% RSLogix 500 project MLO3B JOB 15.RSS, saved by version 10.00.00.00 %
PROJECT "MLO3B"    % processor: Bul.1763 MicroLogix 1100 Series B %

PROGRAM FILES
  LAD 2   15 rungs

DATA FILES
  O0 OUTPUT  4 elements
  I1 INPUT  6 elements
  S2 STATUS  66 elements
  B3 BINARY  1 elements
  T4 TIMER  1 elements
  C5 COUNTER  1 elements
  R6 CONTROL  1 elements
  N7 INTEGER  1 elements
  F8 FLOAT  1 elements

LADDER 2
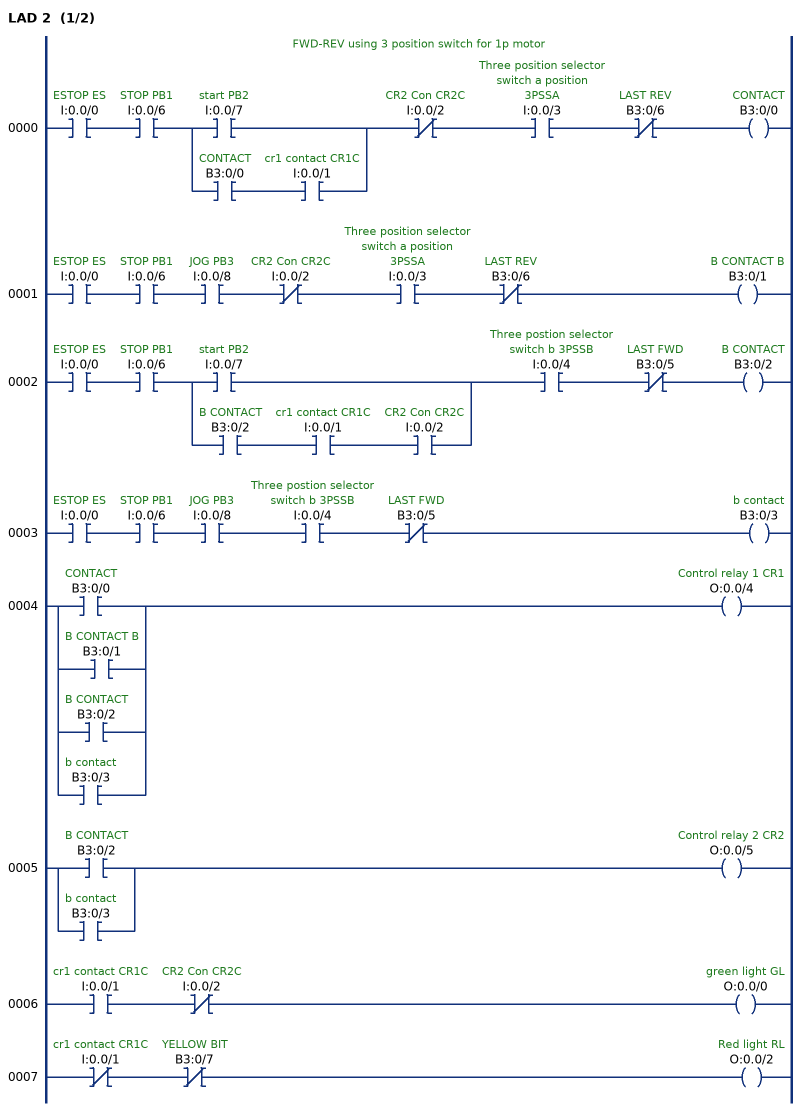
% Rung: 0 %
% FWD-REV using 3 position switch for 1p motor %
SOR XIC I:0.0/0 XIC I:0.0/6 BST XIC I:0.0/7 NXB XIC B3:0/0 XIC I:0.0/1 BND XIO I:0.0/2 XIC I:0.0/3 XIO B3:0/6 OTE B3:0/0 EOR
%   I:0.0/0  ES  "ESTOP" %
%   I:0.0/6  PB1  "STOP" %
%   I:0.0/7  PB2  "start" %
%   B3:0/0  CONTACT %
%   I:0.0/1  CR1C  "cr1 contact" %
%   I:0.0/2  CR2C  "CR2 Con" %
%   I:0.0/3  3PSSA  "Three position selector switch a position" %
%   B3:0/6  "LAST REV" %
% Rung: 1 %
SOR XIC I:0.0/0 XIC I:0.0/6 XIC I:0.0/8 XIO I:0.0/2 XIC I:0.0/3 XIO B3:0/6 OTE B3:0/1 EOR
%   I:0.0/0  ES  "ESTOP" %
%   I:0.0/6  PB1  "STOP" %
%   I:0.0/8  PB3  "JOG" %
%   I:0.0/2  CR2C  "CR2 Con" %
%   I:0.0/3  3PSSA  "Three position selector switch a position" %
%   B3:0/6  "LAST REV" %
%   B3:0/1  B  "B CONTACT" %
% Rung: 2 %
SOR XIC I:0.0/0 XIC I:0.0/6 BST XIC I:0.0/7 NXB XIC B3:0/2 XIC I:0.0/1 XIC I:0.0/2 BND XIC I:0.0/4 XIO B3:0/5 OTE B3:0/2 EOR
%   I:0.0/0  ES  "ESTOP" %
%   I:0.0/6  PB1  "STOP" %
%   I:0.0/7  PB2  "start" %
%   B3:0/2  "B CONTACT" %
%   I:0.0/1  CR1C  "cr1 contact" %
%   I:0.0/2  CR2C  "CR2 Con" %
%   I:0.0/4  3PSSB  "Three postion selector switch b" %
%   B3:0/5  "LAST FWD" %
% Rung: 3 %
SOR XIC I:0.0/0 XIC I:0.0/6 XIC I:0.0/8 XIC I:0.0/4 XIO B3:0/5 OTE B3:0/3 EOR
%   I:0.0/0  ES  "ESTOP" %
%   I:0.0/6  PB1  "STOP" %
%   I:0.0/8  PB3  "JOG" %
%   I:0.0/4  3PSSB  "Three postion selector switch b" %
%   B3:0/5  "LAST FWD" %
%   B3:0/3  "b contact" %
% Rung: 4 %
SOR BST XIC B3:0/0 NXB XIC B3:0/1 NXB XIC B3:0/2 NXB XIC B3:0/3 BND OTE O:0.0/4 EOR
%   B3:0/0  CONTACT %
%   B3:0/1  B  "B CONTACT" %
%   B3:0/2  "B CONTACT" %
%   B3:0/3  "b contact" %
%   O:0.0/4  CR1  "Control relay 1" %
% Rung: 5 %
SOR BST XIC B3:0/2 NXB XIC B3:0/3 BND OTE O:0.0/5 EOR
%   B3:0/2  "B CONTACT" %
%   B3:0/3  "b contact" %
%   O:0.0/5  CR2  "Control relay 2" %
% Rung: 6 %
SOR XIC I:0.0/1 XIO I:0.0/2 OTE O:0.0/0 EOR
%   I:0.0/1  CR1C  "cr1 contact" %
%   I:0.0/2  CR2C  "CR2 Con" %
%   O:0.0/0  GL  "green light" %
% Rung: 7 %
SOR XIO I:0.0/1 XIO B3:0/7 OTE O:0.0/2 EOR
%   I:0.0/1  CR1C  "cr1 contact" %
%   B3:0/7  "YELLOW BIT" %
%   O:0.0/2  RL  "Red light" %

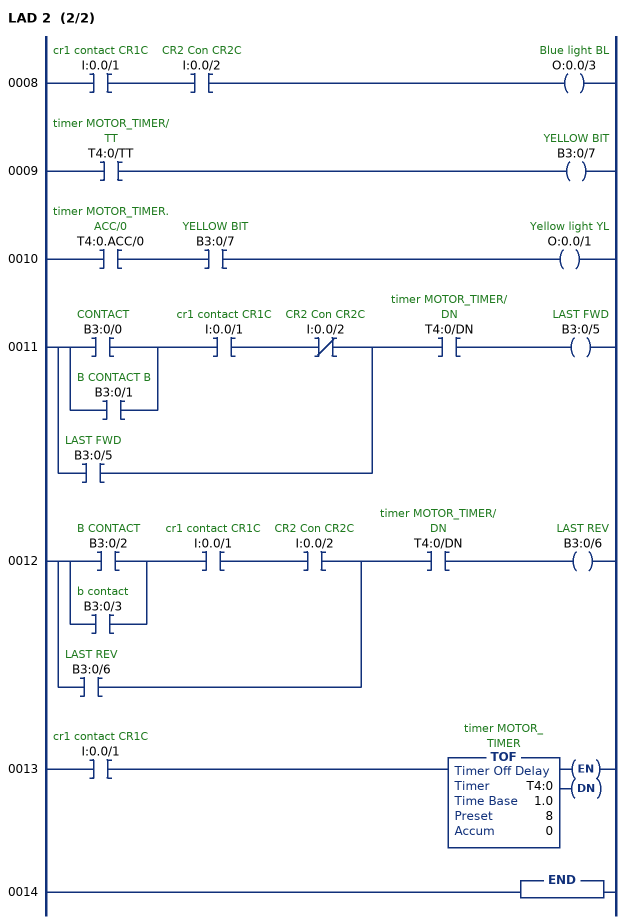
% Rung: 8 %
SOR XIC I:0.0/1 XIC I:0.0/2 OTE O:0.0/3 EOR
%   I:0.0/1  CR1C  "cr1 contact" %
%   I:0.0/2  CR2C  "CR2 Con" %
%   O:0.0/3  BL  "Blue light" %
% Rung: 9 %
SOR XIC T4:0/TT OTE B3:0/7 EOR
%   T4:0  MOTOR_TIMER  "timer" %
%   B3:0/7  "YELLOW BIT" %
% Rung: 10 %
SOR XIC T4:0.ACC/0 XIC B3:0/7 OTE O:0.0/1 EOR
%   T4:0  MOTOR_TIMER  "timer" %
%   B3:0/7  "YELLOW BIT" %
%   O:0.0/1  YL  "Yellow light" %
% Rung: 11 %
SOR BST BST XIC B3:0/0 NXB XIC B3:0/1 BND XIC I:0.0/1 XIO I:0.0/2 NXB XIC B3:0/5 BND XIC T4:0/DN OTE B3:0/5 EOR
%   B3:0/0  CONTACT %
%   B3:0/1  B  "B CONTACT" %
%   I:0.0/1  CR1C  "cr1 contact" %
%   I:0.0/2  CR2C  "CR2 Con" %
%   B3:0/5  "LAST FWD" %
%   T4:0  MOTOR_TIMER  "timer" %
% Rung: 12 %
SOR BST BST XIC B3:0/2 NXB XIC B3:0/3 BND XIC I:0.0/1 XIC I:0.0/2 NXB XIC B3:0/6 BND XIC T4:0/DN OTE B3:0/6 EOR
%   B3:0/2  "B CONTACT" %
%   B3:0/3  "b contact" %
%   I:0.0/1  CR1C  "cr1 contact" %
%   I:0.0/2  CR2C  "CR2 Con" %
%   B3:0/6  "LAST REV" %
%   T4:0  MOTOR_TIMER  "timer" %
% Rung: 13 %
SOR XIC I:0.0/1 TOF T4:0 1.0 8 0 EOR
%   I:0.0/1  CR1C  "cr1 contact" %
%   T4:0  MOTOR_TIMER  "timer" %
% Rung: 14 %
SOR END EOR

OTHER DOCUMENTED ADDRESSES
  GR  "green light"
  GREE  
  I:0.0/5  2PSS  "RUN_JOG"
  IOS  
  O:0.0/6  RED_LIGHT
  O:0.0/7  "Green light"

DATA TABLE (non-zero values as saved)
DATA T4
% .PRE .ACC %
% T4:0 % 8 0
